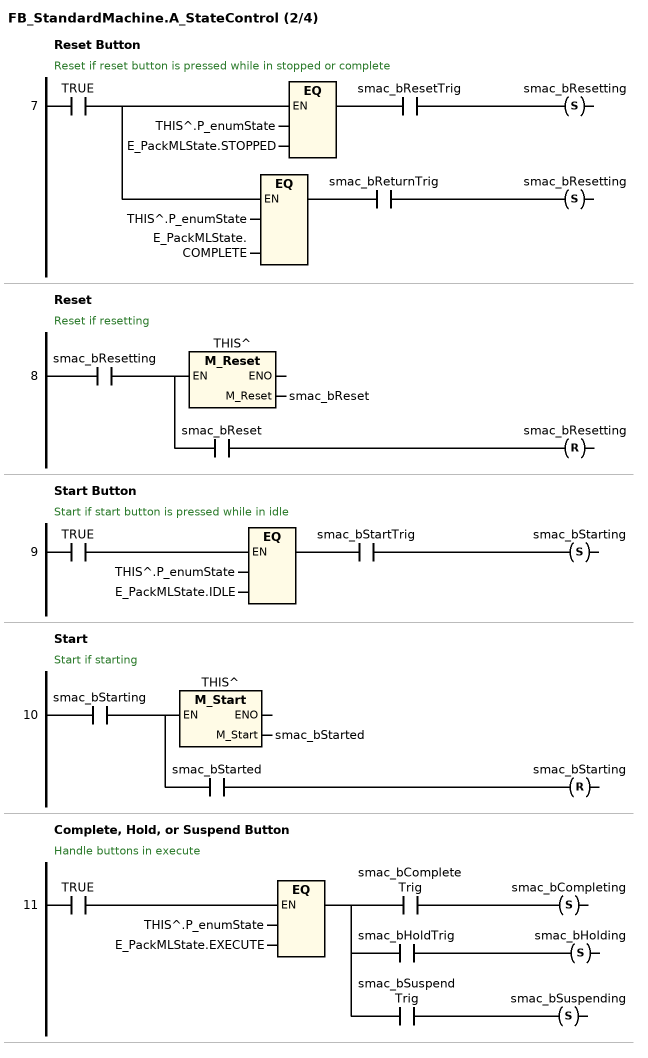
// NETWORK 7: Reset Button
// Reset if reset button is pressed while in stopped or complete
smac_bResetting S= THIS^.P_enumState = E_PackMLState.STOPPED AND smac_bResetTrig;
smac_bResetting S= THIS^.P_enumState = E_PackMLState.COMPLETE AND smac_bReturnTrig;

// NETWORK 8: Reset
// Reset if resetting
_w7 := smac_bResetting;
IF _w7 THEN THIS^.M_Reset(M_Reset => smac_bReset); END_IF
smac_bResetting R= _w7 AND smac_bReset;

// NETWORK 9: Start Button
// Start if start button is pressed while in idle
smac_bStarting S= THIS^.P_enumState = E_PackMLState.IDLE AND smac_bStartTrig;

// NETWORK 10: Start
// Start if starting
_w8 := smac_bStarting;
IF _w8 THEN THIS^.M_Start(M_Start => smac_bStarted); END_IF
smac_bStarting R= _w8 AND smac_bStarted;

// NETWORK 11: Complete, Hold, or Suspend Button
// Handle buttons in execute
_w9 := THIS^.P_enumState = E_PackMLState.EXECUTE;
smac_bCompleting S= _w9 AND smac_bCompleteTrig;
smac_bHolding S= _w9 AND smac_bHoldTrig;
smac_bSuspending S= _w9 AND smac_bSuspendTrig;

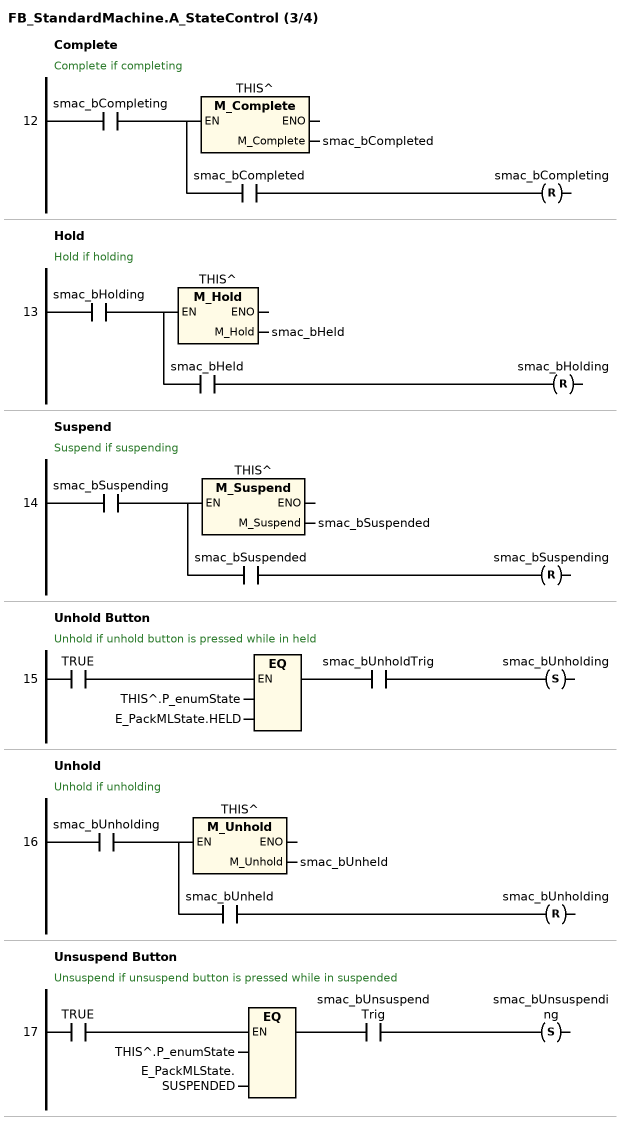
// NETWORK 12: Complete
// Complete if completing
_w10 := smac_bCompleting;
IF _w10 THEN THIS^.M_Complete(M_Complete => smac_bCompleted); END_IF
smac_bCompleting R= _w10 AND smac_bCompleted;

// NETWORK 13: Hold
// Hold if holding
_w11 := smac_bHolding;
IF _w11 THEN THIS^.M_Hold(M_Hold => smac_bHeld); END_IF
smac_bHolding R= _w11 AND smac_bHeld;

// NETWORK 14: Suspend
// Suspend if suspending
_w12 := smac_bSuspending;
IF _w12 THEN THIS^.M_Suspend(M_Suspend => smac_bSuspended); END_IF
smac_bSuspending R= _w12 AND smac_bSuspended;

// NETWORK 15: Unhold Button
// Unhold if unhold button is pressed while in held
smac_bUnholding S= THIS^.P_enumState = E_PackMLState.HELD AND smac_bUnholdTrig;

// NETWORK 16: Unhold
// Unhold if unholding
_w13 := smac_bUnholding;
IF _w13 THEN THIS^.M_Unhold(M_Unhold => smac_bUnheld); END_IF
smac_bUnholding R= _w13 AND smac_bUnheld;

// NETWORK 17: Unsuspend Button
// Unsuspend if unsuspend button is pressed while in suspended
smac_bUnsuspending S= THIS^.P_enumState = E_PackMLState.SUSPENDED AND smac_bUnsuspendTrig;

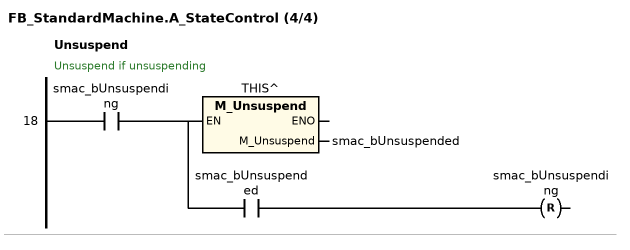
// NETWORK 18: Unsuspend
// Unsuspend if unsuspending
_w14 := smac_bUnsuspending;
IF _w14 THEN THIS^.M_Unsuspend(M_Unsuspend => smac_bUnsuspended); END_IF
smac_bUnsuspending R= _w14 AND smac_bUnsuspended;
END_ACTION

ACTION A_TrackSync:
FOR stdmac_intIndex := 1 TO UINT_TO_INT(GVL_Constants.uintMAX_MACHINE_STATION_COUNT) DO
	// Exit if pointer is not assigned
	IF mac_arrStations[stdmac_intIndex] = 0 THEN
		out_arrStationDesynched[stdmac_intIndex] := FALSE;
		CONTINUE;
	END_IF
	
	// Sync status depends on machine state
	out_arrStationDesynched[stdmac_intIndex] := TRUE;
	stdmac_enumStationState := mac_arrStations[stdmac_intIndex]^.P_enumState;
	stdmac_enumMachineState := THIS^.P_enumState;
	CASE stdmac_enumMachineState OF
		// Aborted, stopped, idle, held, suspended, or completed
		E_PackMLState.ABORTED, E_PackMLState.STOPPED, E_PackMLState.IDLE, 
				E_PackMLState.COMPLETE, E_PackMLState.HELD, E_PackMLState.SUSPENDED:
			IF stdmac_enumStationState = THIS^.P_EnumState THEN
				out_arrStationDesynched[stdmac_intIndex] := FALSE;
			END_IF
			
		// M_Abort
		E_PackMLState.ABORTING:
			CASE stdmac_enumStationState OF
				E_PackMLState.ABORTING, E_PackMLState.ABORTED:
					out_arrStationDesynched[stdmac_intIndex] := FALSE;
			END_CASE
			
		// M_Clear
		E_PackMLState.CLEARING:
			CASE stdmac_enumStationState OF
				E_PackMLState.CLEARING, E_PackMLState.STOPPED:
					out_arrStationDesynched[stdmac_intIndex] := FALSE;
			END_CASE
			
		// M_Stop
		E_PackMLState.STOPPING:
			CASE stdmac_enumStationState OF
				E_PackMLState.STOPPING, E_PackMLState.STOPPED:
					out_arrStationDesynched[stdmac_intIndex] := FALSE;
			END_CASE
			
		// M_Reset
		E_PackMLState.RESETTING:
			CASE stdmac_enumStationState OF
				E_PackMLState.RESETTING, E_PackMLState.IDLE:
					out_arrStationDesynched[stdmac_intIndex] := FALSE;
			END_CASE
			
		// M_Start
		E_PackMLState.STARTING:
			CASE stdmac_enumStationState OF
				E_PackMLState.STARTING, E_PackMLState.EXECUTE, E_PackMLState.HOLDING,
						E_PackMLState.HELD, E_PackMLState.UNHOLDING, E_PackMLState.SUSPENDING,
						E_PackMLState.SUSPENDED, E_PackMLState.UNSUSPENDING:
					out_arrStationDesynched[stdmac_intIndex] := FALSE;
			END_CASE
			
		// Execute
		E_PackMLState.EXECUTE:
			CASE stdmac_enumStationState OF
				E_PackMLState.EXECUTE, E_PackMLState.HOLDING, E_PackMLState.HELD,
						E_PackMLState.UNHOLDING, E_PackMLState.SUSPENDING,
						E_PackMLState.SUSPENDED, E_PackMLState.UNSUSPENDING:
					out_arrStationDesynched[stdmac_intIndex] := FALSE;
			END_CASE
			
		// M_Complete
		E_PackMLState.COMPLETING:
			CASE stdmac_enumStationState OF
				E_PackMLState.COMPLETING, E_PackMLState.COMPLETE:
					out_arrStationDesynched[stdmac_intIndex] := FALSE;
			END_CASE
			
		// M_Hold
		E_PackMLState.HOLDING:
			CASE stdmac_enumStationState OF
				E_PackMLState.HOLDING, E_PackMLState.HELD:
					out_arrStationDesynched[stdmac_intIndex] := FALSE;
			END_CASE
			
		// M_Unhold
		E_PackMLState.UNHOLDING:
			CASE stdmac_enumStationState OF
				E_PackMLState.EXECUTE, E_PackMLState.HOLDING, E_PackMLState.HELD,
						E_PackMLState.UNHOLDING, E_PackMLState.SUSPENDING,
						E_PackMLState.SUSPENDED, E_PackMLState.UNSUSPENDING:
					out_arrStationDesynched[stdmac_intIndex] := FALSE;
			END_CASE
			
		// M_Suspend
		E_PackMLState.SUSPENDING:
			CASE stdmac_enumStationState OF
				E_PackMLState.SUSPENDING, E_PackMLState.SUSPENDED:
					out_arrStationDesynched[stdmac_intIndex] := FALSE;
			END_CASE
			
		// M_Unsuspend
		E_PackMLState.UNSUSPENDING:
			CASE stdmac_enumStationState OF
				E_PackMLState.EXECUTE, E_PackMLState.HOLDING, E_PackMLState.HELD,
						E_PackMLState.UNHOLDING, E_PackMLState.SUSPENDING,
						E_PackMLState.SUSPENDED, E_PackMLState.UNSUSPENDING:
					out_arrStationDesynched[stdmac_intIndex] := FALSE;
			END_CASE
	END_CASE
END_FOR
END_ACTION

END_FUNCTION_BLOCK

// Interfaces/Stations/I_UserControls
INTERFACE I_UserControls

(* Clears the user prompt outputs. *)
METHOD M_ClearUserPrompt : BOOL
VAR_INPUT
END_VAR
END_METHOD

(* Sets user prompt based on given code, and awaits user input. *)
METHOD M_HandleException : BOOL
VAR_INPUT
	(* Prompt code for the exception message. *)
	_in_udintPromptCode: UDINT;
	(* Error code to set in case user aborts. *)
	_in_udintErrorCode: UDINT;
END_VAR
VAR_OUTPUT
END_VAR
END_METHOD

(* Sets out_strUserPromptCode and out_strUserPromptMessage based on
	the given user prompt code. *)
METHOD M_SetUserPrompt : BOOL
VAR_INPUT
	(* Prompt code to use for this user prompt. *)
	_in_udintCode: UDINT;
END_VAR
END_METHOD

END_INTERFACE

// Concrete/Stations/Device Test Station/FB_DeviceTestStation
FUNCTION_BLOCK FB_DeviceTestStation EXTENDS FB_SimpleStation
VAR_INPUT
	ref_fbDevice: REFERENCE TO FB_Device; // The device to be tested

	in_strProgram: T_MaxString; // Program to load when testing program loading
END_VAR
VAR_OUTPUT
	out_bAbortTested: BOOL; // Gets set to TRUE once M_Abort on ref_fbDevice has been tested once
	
	out_bConnectTested: BOOL;  // Gets set to TRUE once M_Connect on ref_fbDevice has been tested once
	out_bDisconnectTested: BOOL;  // Gets set to TRUE once M_Disconnect on ref_fbDevice has been tested once
	
	out_bEnableTested: BOOL; // Gets set to TRUE once M_Enable on ref_fbDevice has been tested once
	out_bDisableTested: BOOL; // Gets set to TRUE once M_Disable on ref_fbDevice has been tested once
	
	out_bPowerOnTested: BOOL; // Gets set to TRUE once M_PowerOn on ref_fbDevice has been tested once
	out_bPowerOffTested: BOOL; // Gets set to TRUE once M_PowerOff on ref_fbDevice has been tested once
	
	out_bLoadProgramTested: BOOL; // Gets set to TRUE once M_LoadProgram on ref_fbDevice has been tested once
	out_bStartProgramTested: BOOL; // Gets set to TRUE once M_StartProgram on ref_fbDevice has been tested once
	out_bStopProgramTested: BOOL; // Gets set to TRUE once M_StopProgram on ref_fbDevice has been tested once
	out_bPauseProgramTested: BOOL; // Gets set to TRUE once M_PauseProgram on ref_fbDevice has been tested once
	out_bUnpauseProgramTested: BOOL; // Gets set to TRUE once M_StartProgram on ref_fbDevice has been tested once after M_PauseProgram was used
	out_bStopPausedProgramTested: BOOL; // Gets set to TRUE once M_StopProgram on ref_fbDevice has been tested once after M_PauseProgram was used
	
	out_bResetTested: BOOL; // Gets set to TRUE once M_Reset on ref_fbDevice has been tested once
END_VAR
VAR
	bDeviceReset: BOOL;
	
	bDeviceConnected: BOOL;
	bDeviceDisconnected: BOOL;
	
	bDevicePoweredOn: BOOL;
	bDevicePoweredOff: BOOL;
	
	bDeviceEnabled: BOOL;
	bDeviceDisabled: BOOL;
	
	bDeviceProgramLoaded: BOOL;
	bDeviceProgramStarted: BOOL;
	bDeviceProgramStopped: BOOL;
	bDeviceProgramPaused: BOOL;

	// Device test trackers
	fbDeviceAborted: R_TRIG;
	fbDeviceReset: F_TRIG;
	fbDeviceConnected: R_TRIG;
	fbDeviceDisconnected: F_TRIG;
	fbDeviceEnabled: R_TRIG;
	fbDeviceDisabled: F_TRIG;
	fbDevicePoweredOn: R_TRIG;
	fbDevicePoweredOff: F_TRIG;
	fbDeviceProgramLoaded: R_TRIG;
	enumLastState: E_ProgramState;
END_VAR

THIS^.M_SetDevice(1, ref_fbDevice);

A_RunSimpleStation();

A_DeviceTestTracking();

ACTION A_DeviceTestTracking:
// Check device error state
fbDeviceAborted(CLK:=ref_fbDevice.P_bError);
fbDeviceReset(CLK:=ref_fbDevice.P_bError);

// Check device connection state
fbDeviceConnected(CLK:=ref_fbDevice.P_bConnected);
fbDeviceDisconnected(CLK:=ref_fbDevice.P_bConnected);

// Check device enable state
fbDeviceEnabled(CLK:=ref_fbDevice.P_bEnabled);
fbDeviceDisabled(CLK:=ref_fbDevice.P_bEnabled);

// Check device power state
fbDevicePoweredOn(CLK:=ref_fbDevice.P_bPoweredOn);
fbDevicePoweredOff(CLK:=ref_fbDevice.P_bPoweredOn);

// Check device program load state
fbDeviceProgramLoaded(CLK:=(
	ref_fbDevice.P_strCurrentProgram = in_strProgram
	AND LEN(in_strProgram) > 0));
	
// Set outputs based on triggers
IF fbDeviceAborted.Q		THEN out_bAbortTested 		:= TRUE; END_IF
IF fbDeviceReset.Q			THEN out_bResetTested 		:= TRUE; END_IF
IF fbDeviceConnected.Q		THEN out_bConnectTested 	:= TRUE; END_IF
IF fbDeviceDisconnected.Q	THEN out_bDisconnectTested	:= TRUE; END_IF
IF fbDeviceEnabled.Q		THEN out_bEnableTested 		:= TRUE; END_IF
IF fbDeviceDisabled.Q		THEN out_bDisableTested 	:= TRUE; END_IF
IF fbDevicePoweredOn.Q		THEN out_bPowerOnTested 	:= TRUE; END_IF
IF fbDevicePoweredOff.Q		THEN out_bPowerOffTested 	:= TRUE; END_IF
IF fbDeviceProgramLoaded.Q	THEN out_bLoadProgramTested	:= TRUE; END_IF

// Set program control state outputs
IF enumLastState = E_ProgramState.Stopped THEN
	IF ref_fbDevice.P_enumProgramState = E_ProgramState.Running THEN
		out_bStartProgramTested := TRUE;
	END_IF
ELSIF enumLastState = E_ProgramState.Running THEN
	IF ref_fbDevice.P_enumProgramState = E_ProgramState.Stopped THEN
		out_bStopProgramTested := TRUE;
	ELSIF ref_fbDevice.P_enumProgramState = E_ProgramState.Paused THEN
		out_bPauseProgramTested := TRUE;
	END_IF
ELSIF enumLastState = E_ProgramState.Paused THEN
	IF ref_fbDevice.P_enumProgramState = E_ProgramState.Running THEN
		out_bUnpauseProgramTested := TRUE;
	ELSIF ref_fbDevice.P_enumProgramState = E_ProgramState.Stopped THEN
		out_bStopPausedProgramTested := TRUE;
	END_IF
END_IF
enumLastState := ref_fbDevice.P_enumProgramState;
END_ACTION

END_FUNCTION_BLOCK

// Concrete/Stations/Simple Station/FB_SimpleStation
(*
	Simple station that extends adds buttons to FB_Station
*)
{attribute 'hide_all_locals'}
FUNCTION_BLOCK FB_SimpleStation EXTENDS FB_Station
VAR_INPUT
	(* Immediately abort all stations from whatever state they are in and
		go to the Aborted state. *)
	in_bAbortBtn : BOOL;
	(* Immediately stop all stations from whatever state they are in and
		go to the Stopped state. *)
	in_bStopBtn : BOOL;
	(* Clear all stations from the Aborted state and go to the Stopped state. *)
	in_bClearBtn : BOOL;
	(* Reset all stations from the Stopped state and go to the Idle state. *)
	in_bResetBtn : BOOL;
	(* Start all stations from the Idle state and go to the Execute state. *)
	in_bStartBtn : BOOL;
	(* Hold all stations from the Execute state and go to the Held state. *)
	in_bHoldBtn : BOOL;
	(* Unhold all stations from the Held state and go to the Execute state. *)
	in_bUnholdBtn : BOOL;
	(* Suspend all stations from the Execute state and go to the Held Suspended. *)
	in_bSuspendBtn : BOOL;
	(* Unsuspend all stations from the Suspended state and go to the Execute state. *)
	in_bUnsuspendBtn : BOOL;
	(* Complete all stations from the Execute state and go to the Completed state. *)
	in_bCompleteBtn : BOOL;
	(* Return all stations from the Completed state and go to the Idle state. *)
	in_bReturnBtn : BOOL;
END_VAR
VAR_OUTPUT
END_VAR
VAR
	// Abort
	ssta_fbAbortTrig: R_TRIG;
	ssta_bAbortTrig: BOOL;
	ssta_bAborting: BOOL;
	ssta_bAborted: BOOL;

	// Stop
	ssta_fbStopTrig: R_TRIG;
	ssta_bStopTrig: BOOL;
	ssta_bStopping: BOOL;
	ssta_bStopped: BOOL;
	
	// Aborted
	ssta_fbClearTrig: R_TRIG;
	ssta_bClearTrig: BOOL;
	
	// Stopped
	ssta_fbResetTrig: R_TRIG;
	ssta_bResetTrig: BOOL;
	
	// Idle
	ssta_fbStartTrig: R_TRIG;
	ssta_bStartTrig: BOOL;
	
	// Execute
	ssta_fbCompleteTrig: R_TRIG;
	ssta_bCompleteTrig: BOOL;
	ssta_fbHoldTrig: R_TRIG;
	ssta_bHoldTrig: BOOL;
	ssta_fbSuspendTrig: R_TRIG;
	ssta_bSuspendTrig: BOOL;
	
	// Complete
	ssta_fbReturnTrig: R_TRIG;
	ssta_bReturnTrig: BOOL;
	
	// Held
	ssta_fbUnholdTrig: R_TRIG;
	ssta_bUnholdTrig: BOOL;
	
	// Suspended
	ssta_fbUnsuspendTrig: R_TRIG;
	ssta_bUnsuspendTrig: BOOL;
END_VAR

THIS^.A_RunSimpleStation();

ACTION A_Buttons:
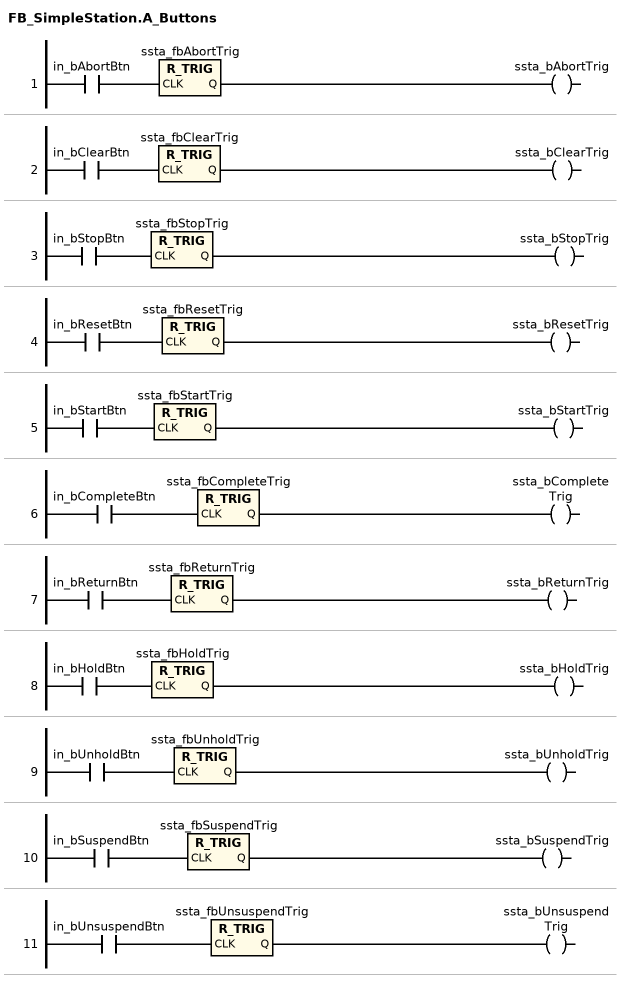
// NETWORK 1
ssta_fbAbortTrig(CLK := in_bAbortBtn); // R_TRIG
ssta_bAbortTrig := ssta_fbAbortTrig.Q;

// NETWORK 2
ssta_fbClearTrig(CLK := in_bClearBtn); // R_TRIG
ssta_bClearTrig := ssta_fbClearTrig.Q;

// NETWORK 3
ssta_fbStopTrig(CLK := in_bStopBtn); // R_TRIG
ssta_bStopTrig := ssta_fbStopTrig.Q;

// NETWORK 4
ssta_fbResetTrig(CLK := in_bResetBtn); // R_TRIG
ssta_bResetTrig := ssta_fbResetTrig.Q;

// NETWORK 5
ssta_fbStartTrig(CLK := in_bStartBtn); // R_TRIG
ssta_bStartTrig := ssta_fbStartTrig.Q;

// NETWORK 6
ssta_fbCompleteTrig(CLK := in_bCompleteBtn); // R_TRIG
ssta_bCompleteTrig := ssta_fbCompleteTrig.Q;

// NETWORK 7
ssta_fbReturnTrig(CLK := in_bReturnBtn); // R_TRIG
ssta_bReturnTrig := ssta_fbReturnTrig.Q;

// NETWORK 8
ssta_fbHoldTrig(CLK := in_bHoldBtn); // R_TRIG
ssta_bHoldTrig := ssta_fbHoldTrig.Q;

// NETWORK 9
ssta_fbUnholdTrig(CLK := in_bUnholdBtn); // R_TRIG
ssta_bUnholdTrig := ssta_fbUnholdTrig.Q;

// NETWORK 10
ssta_fbSuspendTrig(CLK := in_bSuspendBtn); // R_TRIG
ssta_bSuspendTrig := ssta_fbSuspendTrig.Q;

// NETWORK 11
ssta_fbUnsuspendTrig(CLK := in_bUnsuspendBtn); // R_TRIG
ssta_bUnsuspendTrig := ssta_fbUnsuspendTrig.Q;
END_ACTION

ACTION A_RunSimpleStation:
THIS^.A_StopAndAbort();
THIS^.A_Buttons();
THIS^.A_StateMachine();
END_ACTION

ACTION A_StopAndAbort:
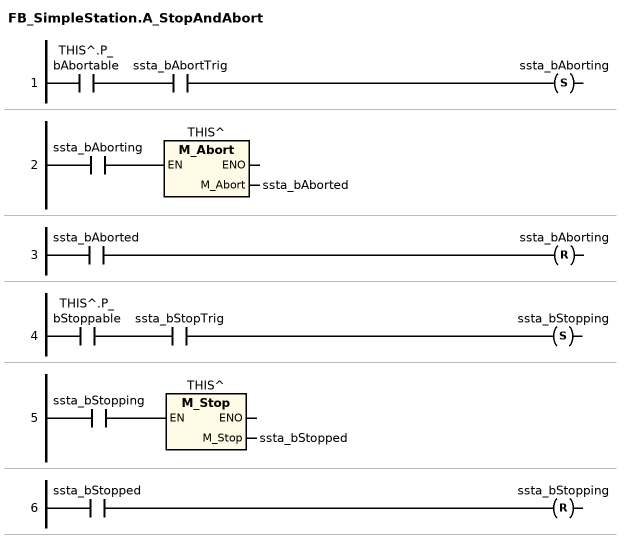
// NETWORK 1
ssta_bAborting S= THIS^.P_bAbortable AND ssta_bAbortTrig;

// NETWORK 2
IF ssta_bAborting THEN THIS^.M_Abort(M_Abort => ssta_bAborted); END_IF

// NETWORK 3
ssta_bAborting R= ssta_bAborted;

// NETWORK 4
ssta_bStopping S= THIS^.P_bStoppable AND ssta_bStopTrig;

// NETWORK 5
IF ssta_bStopping THEN THIS^.M_Stop(M_Stop => ssta_bStopped); END_IF

// NETWORK 6
ssta_bStopping R= ssta_bStopped;
END_ACTION

(* This state is entered after the aborting state completes, and should
not modify anything in the module while awaiting an explicit 'Clear' command. *)
METHOD M011_Aborted : BOOL
VAR_OUTPUT
	(* This should be set to true once an explicit 'Clear' command is received.
	Once set to true, the state machine will move to the 'Clearing' state. *)
	bClear	: BOOL;
END_VAR
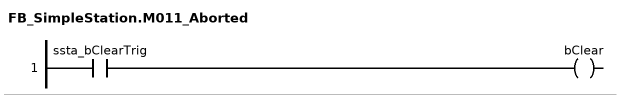
// NETWORK 1
bClear := ssta_bClearTrig;
END_METHOD

(* The machine should be stationary and awaiting an explicit 'Reset' command
while in this state. Once the 'Reset' command is received, the state machine
will move to the 'Resetting' state. *)
METHOD M111_Stopped : BOOL
VAR_OUTPUT
	(* This should be set to true if an explicit reset command is received.
	Once set to true, the state machine will move to the 'Resetting' state. *)
	bReset	: BOOL;
	(* This should be set to true if a potentially hazardous error or a safety
	fault has occurred in any tasks. Once set to true, the state machine will
	move to the 'Aborting' state. *)
	bAbort	: BOOL;
END_VAR
VAR
	_bDeviceError: BOOL;
	_strDeviceErrorId: T_MaxString;
	_udintDeviceErrorCode: UDINT;
	_strDeviceErrorMsg: T_MaxString;
	_strErrorMsg: STRING(255);
END_VAR
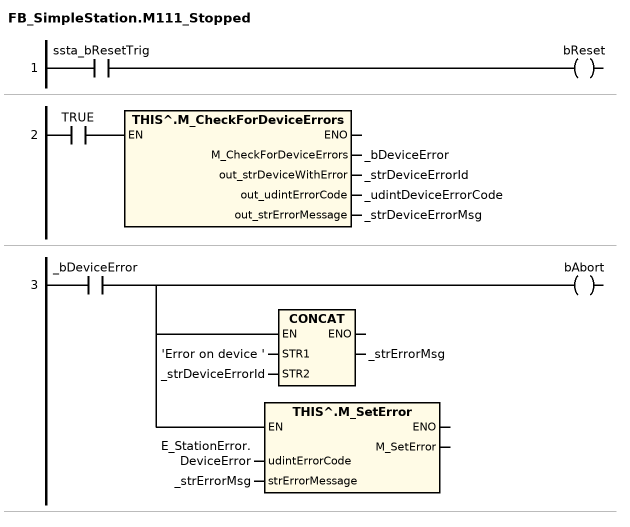
// NETWORK 1
bReset := ssta_bResetTrig;

// NETWORK 2
_bDeviceError := THIS^.M_CheckForDeviceErrors(out_strDeviceWithError => _strDeviceErrorId, out_udintErrorCode => _udintDeviceErrorCode, out_strErrorMessage => _strDeviceErrorMsg);

// NETWORK 3
bAbort := _bDeviceError;
IF _bDeviceError THEN _strErrorMsg := CONCAT(STR1 := 'Error on device ', STR2 := _strDeviceErrorId); END_IF
IF _bDeviceError THEN
    THIS^.M_SetError(udintErrorCode := E_StationError.DeviceError, strErrorMessage := _strErrorMsg);
END_IF
END_METHOD

(* This state should maintain the status of the module and its components that
was set by the resetting step while awaiting an explicit 'Start' command. *)
METHOD M211_Idle : BOOL
VAR_OUTPUT
	(* This should be set to true if an explicit 'Start' command is received.
	Once set to true, the state machine will move to the 'Starting' state. *)
	bStart	: BOOL;
	(* This should be set to true if an external source requests that the module
	exit its current state and come to a controlled stop. Once set to true, the
	state machine will move to the 'Stopping' state. *)
	bStop	: BOOL;
	(* This should be set to true if a potentially hazardous error or a safety
	fault has occurred in any tasks. Once set to true, the state machine will
	move to the 'Aborting' state. *)
	bAbort	: BOOL;
END_VAR
VAR
	_bDeviceError: BOOL;
	_strDeviceErrorId: T_MaxString;
	_udintDeviceErrorCode: UDINT;
	_strDeviceErrorMsg: T_MaxString;
	_strErrorMsg: STRING(255);
END_VAR
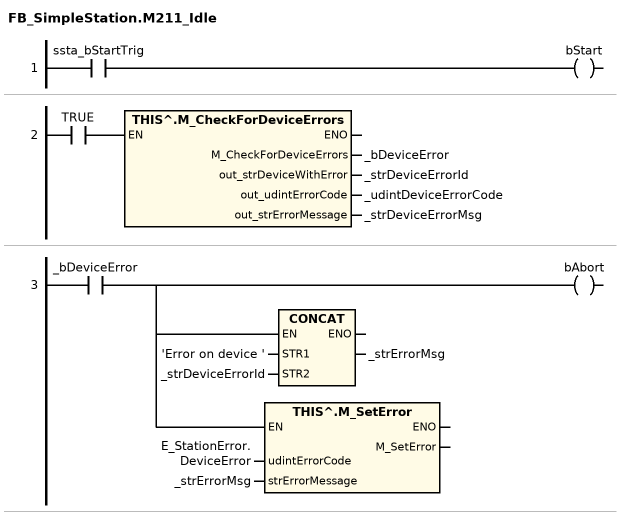
// NETWORK 1
bStart := ssta_bStartTrig;

// NETWORK 2
_bDeviceError := THIS^.M_CheckForDeviceErrors(out_strDeviceWithError => _strDeviceErrorId, out_udintErrorCode => _udintDeviceErrorCode, out_strErrorMessage => _strDeviceErrorMsg);

// NETWORK 3
bAbort := _bDeviceError;
IF _bDeviceError THEN _strErrorMsg := CONCAT(STR1 := 'Error on device ', STR2 := _strDeviceErrorId); END_IF
IF _bDeviceError THEN
    THIS^.M_SetError(udintErrorCode := E_StationError.DeviceError, strErrorMessage := _strErrorMsg);
END_IF
END_METHOD

(* The module should remain in this state while it is actively performing
automated tasks. Once all work is finished the state machine should move to the
'Completing' state. *)
METHOD M311_Execute : BOOL
VAR_OUTPUT
	(* This should be set to true once all tasks are complete and automated
	execution should be ended. Once set to true, the state machine will move to
	the 'Completing' state. *)
	bFinished	: BOOL;
	(* This should be set to true as a result of an explicit 'Hold' command
	or if internal conditions require the module to stop operation without
	completely exiting the execution sequence. Once set to true, the state
	machine will move to the 'Holding' state. *)
	bHold	: BOOL;
	(* This should be set to true if external conditions require the module to
	suspend operation until the external conditions are cleared. Once set to
	true, the state machine will move to the 'Suspending' state. *)
	bSuspend	: BOOL;
	(* This should be set to true if an external source requests that the module
	exit its current state and come to a controlled stop. Once set to true, the
	state machine will move to the 'Stopping' state. *)
	bStop	: BOOL;
	(* This should be set to true if a potentially hazardous error or a safety
	fault has occurred in any tasks. Once set to true, the state machine will
	move to the 'Aborting' state. *)
	bAbort	: BOOL;
END_VAR
VAR
	_bDeviceError: BOOL;
	_strDeviceErrorId: T_MaxString;
	_udintDeviceErrorCode: UDINT;
	_strDeviceErrorMsg: T_MaxString;
	_strErrorMsg: STRING(255);
END_VAR
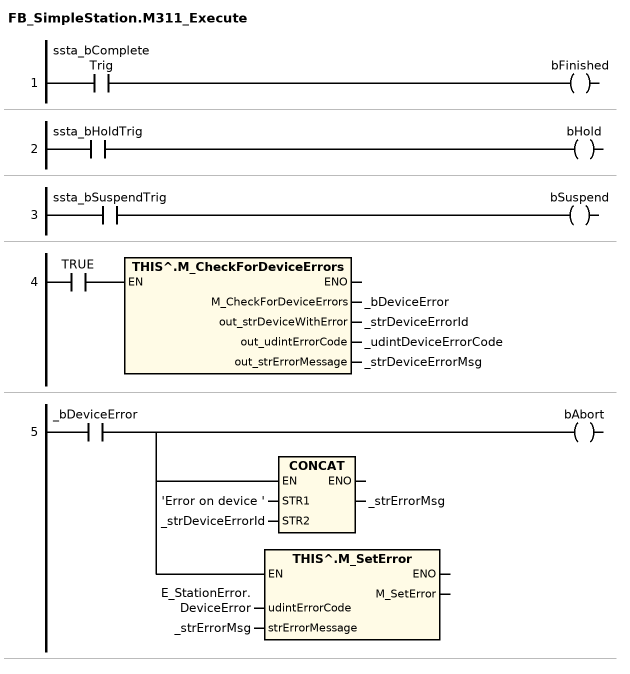
// NETWORK 1
bFinished := ssta_bCompleteTrig;

// NETWORK 2
bHold := ssta_bHoldTrig;

// NETWORK 3
bSuspend := ssta_bSuspendTrig;

// NETWORK 4
_bDeviceError := THIS^.M_CheckForDeviceErrors(out_strDeviceWithError => _strDeviceErrorId, out_udintErrorCode => _udintDeviceErrorCode, out_strErrorMessage => _strDeviceErrorMsg);

// NETWORK 5
bAbort := _bDeviceError;
IF _bDeviceError THEN _strErrorMsg := CONCAT(STR1 := 'Error on device ', STR2 := _strDeviceErrorId); END_IF
IF _bDeviceError THEN
    THIS^.M_SetError(udintErrorCode := E_StationError.DeviceError, strErrorMessage := _strErrorMsg);
END_IF
END_METHOD

(* The module should remain stationary within this state while maintaing any
execution statistics and awaiting an explicit 'Return' command. *)
METHOD M331_Complete : BOOL
VAR_OUTPUT
	(* This should be set to true if an explicit 'Return' command is received.
	Once set to true, the state machine will move to the 'Resetting' state. *)
	bReturn	: BOOL;
	(* This should be set to true if an external source requests that the module
	exit its current state and come to a controlled stop. Once set to true, the
	state machine will move to the 'Stopping' state. *)
	bStop	: BOOL;
	(* This should be set to true if a potentially hazardous error or a safety
	fault has occurred in any tasks. Once set to true, the state machine will
	move to the 'Aborting' state. *)
	bAbort	: BOOL;
END_VAR
VAR
	_bDeviceError: BOOL;
	_strDeviceErrorId: T_MaxString;
	_udintDeviceErrorCode: UDINT;
	_strDeviceErrorMsg: T_MaxString;
	_strErrorMsg: STRING(255);
END_VAR
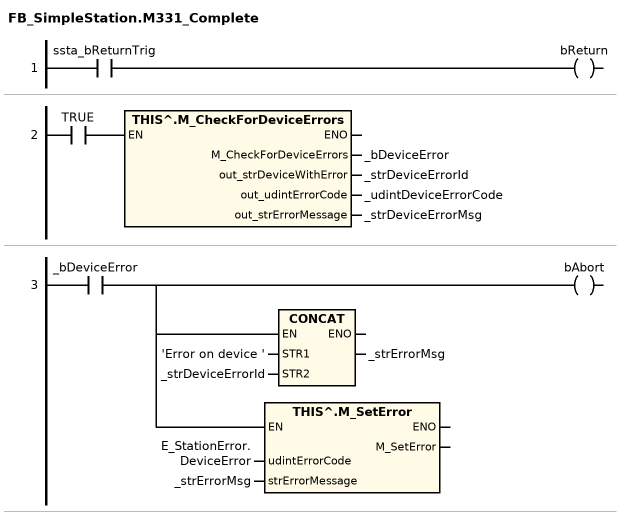
// NETWORK 1
bReturn := ssta_bReturnTrig;

// NETWORK 2
_bDeviceError := THIS^.M_CheckForDeviceErrors(out_strDeviceWithError => _strDeviceErrorId, out_udintErrorCode => _udintDeviceErrorCode, out_strErrorMessage => _strDeviceErrorMsg);

// NETWORK 3
bAbort := _bDeviceError;
IF _bDeviceError THEN _strErrorMsg := CONCAT(STR1 := 'Error on device ', STR2 := _strDeviceErrorId); END_IF
IF _bDeviceError THEN
    THIS^.M_SetError(udintErrorCode := E_StationError.DeviceError, strErrorMessage := _strErrorMsg);
END_IF
END_METHOD

(* In this state the most recent execution status should be maintained while
awaiting an explicit 'Unhold' command once internal conditions are satisfactory. *)
METHOD M411_Held : BOOL
VAR_OUTPUT
	(* This should be set to true if an explicit 'Unhold' command is received.
	Once set to true, the state machine will move to the 'Unholding' state. *)
	bUnhold	: BOOL;
	(* This should be set to true if an external source requests that the module
	exit its current state and come to a controlled stop. Once set to true, the
	state machine will move to the 'Stopping' state. *)
	bStop	: BOOL;
	(* This should be set to true if a potentially hazardous error or a safety
	fault has occurred in any tasks. Once set to true, the state machine will
	move to the 'Aborting' state. *)
	bAbort	: BOOL;
END_VAR
VAR
	_bDeviceError: BOOL;
	_strDeviceErrorId: T_MaxString;
	_udintDeviceErrorCode: UDINT;
	_strDeviceErrorMsg: T_MaxString;
	_strErrorMsg: STRING(255);
END_VAR
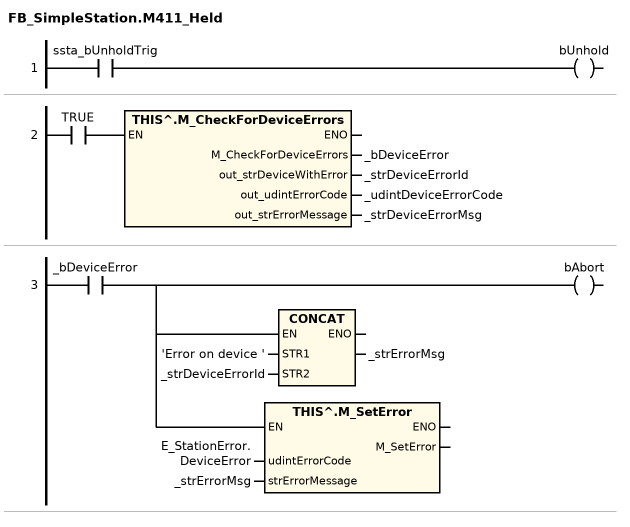
// NETWORK 1
bUnhold := ssta_bUnholdTrig;

// NETWORK 2
_bDeviceError := THIS^.M_CheckForDeviceErrors(out_strDeviceWithError => _strDeviceErrorId, out_udintErrorCode => _udintDeviceErrorCode, out_strErrorMessage => _strDeviceErrorMsg);

// NETWORK 3
bAbort := _bDeviceError;
IF _bDeviceError THEN _strErrorMsg := CONCAT(STR1 := 'Error on device ', STR2 := _strDeviceErrorId); END_IF
IF _bDeviceError THEN
    THIS^.M_SetError(udintErrorCode := E_StationError.DeviceError, strErrorMessage := _strErrorMsg);
END_IF
END_METHOD

(* In this state the most recent execution status should be maintained while
awaiting an explicit 'Unsuspend' command once external conditions are satisfactory. *)
METHOD M511_Suspended : BOOL
VAR_OUTPUT
	(* This should be set to true if an explicit 'Unsuspend' command is received.
	Once set to true, the state machine will move to the 'Unsuspending' state. *)
	bUnsuspend	: BOOL;
	(* This should be set to true if an external source requests that the module
	exit its current state and come to a controlled stop. Once set to true, the
	state machine will move to the 'Stopping' state. *)
	bStop	: BOOL;
	(* This should be set to true if a potentially hazardous error or a safety
	fault has occurred in any tasks. Once set to true, the state machine will
	move to the 'Aborting' state. *)
	bAbort	: BOOL;
END_VAR
VAR
	_bDeviceError: BOOL;
	_strDeviceErrorId: T_MaxString;
	_udintDeviceErrorCode: UDINT;
	_strDeviceErrorMsg: T_MaxString;
	_strErrorMsg: STRING(255);
END_VAR
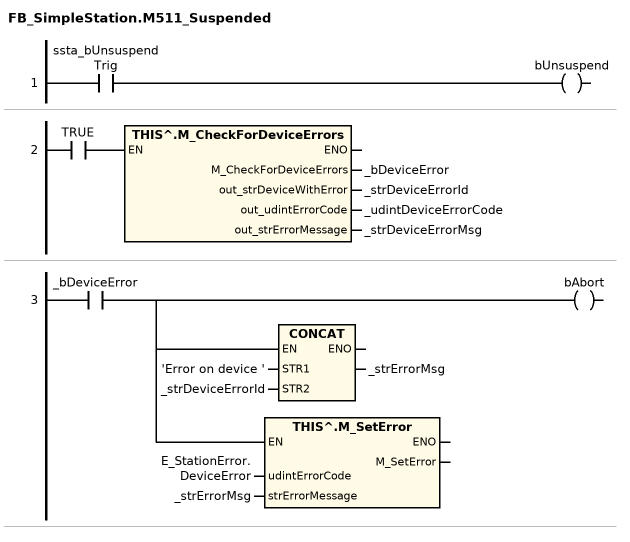
// NETWORK 1
bUnsuspend := ssta_bUnsuspendTrig;

// NETWORK 2
_bDeviceError := THIS^.M_CheckForDeviceErrors(out_strDeviceWithError => _strDeviceErrorId, out_udintErrorCode => _udintDeviceErrorCode, out_strErrorMessage => _strDeviceErrorMsg);

// NETWORK 3
bAbort := _bDeviceError;
IF _bDeviceError THEN _strErrorMsg := CONCAT(STR1 := 'Error on device ', STR2 := _strDeviceErrorId); END_IF
IF _bDeviceError THEN
    THIS^.M_SetError(udintErrorCode := E_StationError.DeviceError, strErrorMessage := _strErrorMsg);
END_IF
END_METHOD

END_FUNCTION_BLOCK

// Concrete/Stations/Remote Machine Station/FB_RemoteMachineStation
(* Function block for running a remote machine as a standard station.
	Make sure to call A_RunRemoteMachine(), which calls A_StateMachine() *)
FUNCTION_BLOCK FB_RemoteMachineStation EXTENDS FB_StandardStation 
	IMPLEMENTS I_SimpleTransitionStatesOnly, I_RemoteCycleControls
VAR CONSTANT
	rms_timeCHECK_TIME: TIME := T#1S;
	rms_timeCHECK_WAIT_TIME: TIME := T#100MS;
	rms_timeSYNC_TIME: TIME := T#1S;
END_VAR
VAR_INPUT
	(* Current remote machine state. *)
	in_enumRemoteMachineState: E_PackMLState;
	(* Remote machine error. *)
	in_bRemoteError: BOOL;
	(* Remote machine error code. *)
	in_udintRemoteErrorCode: UDINT;
	(* Ready to run signal from the remote machine. *)
	in_bRemoteReadyToRun: BOOL;
	(* Check value set by the remote machine. *)
	in_bRemoteCheckResponse: BOOL;
END_VAR
VAR_OUTPUT
	(* Run cycle command to be sent to the remote machine. *)
	out_bRemoteRunCycleCommand: BOOL;
	(* Struct of remote machine state change commands. *)
	out_stRemoteMachineCommands: ST_PackMLStateCommands;
	(* The remote machine should set in_bRemoteCheckResponse to this value to
		verify connection. *)
	out_bRemoteCheck: BOOL;
	(* TRUE if the remote machine is connected based on the remote check sequence. *)
	out_bRemoteConnected: BOOL;
END_VAR
VAR	
	rms_intRemoteCheckStep: INT;
	rms_fbCheckTimer: TON;
	rms_fbCheckWaitTimer: TON;
	rms_fbSyncTimer: TON;
	rms_enumRemoteMachineState: E_PackMLState;
	rms_enumStationState: E_PackMLState;
	rms_bRemoteMachineDesynched: BOOL;
END_VAR

A_RunRemoteMachine();

(* If the remote is ready to run, returns TRUE. *)
METHOD M_AwaitRemoteCycleEnd : BOOL
IF NOT in_bRemoteReadyToRun THEN
	out_bRemoteRunCycleCommand := FALSE;
ELSE
	M_AwaitRemoteCycleEnd := TRUE;
END_IF
END_METHOD

(* Sets run cycle command to TRUE and then waits for either the remote
	ready to run signal to get reset or for the remote to be awaiting
	end, which can happen if the remote cycle time is quicker than the
	main machine. *)
METHOD M_AwaitRemoteCycleStart : BOOL
IF in_bRemoteReadyToRun THEN
	out_bRemoteRunCycleCommand := TRUE;
ELSE
	M_AwaitRemoteCycleStart := TRUE;
END_IF
END_METHOD

METHOD M_ResetRemoteCycle : BOOL
out_bRemoteRunCycleCommand := FALSE;
END_METHOD

(* The 'Aborting' state can be entered at any time while within the 'abortable'
section of the state machine. It is typically entered in response to an 'Abort'
command or a critical fault. The logic should safely but rapidly bring the
components of the module to a stop while maintaining as much information about
the pre-abort scenario as possible. *)
METHOD M001_Aborting : BOOL
VAR_OUTPUT
	(* This should be set to true once all components of the module have safely
	come to a stop. Once set to true, the state machine will move to the
	'Aborted' state. *)
	bAborted	: BOOL;
END_VAR

VAR
	_rms_bAborted: BOOL;
END_VAR
VAR_INST // added by the converter: edge detectors and wires of the graphical bodies
    _w1 : BOOL;
END_VAR
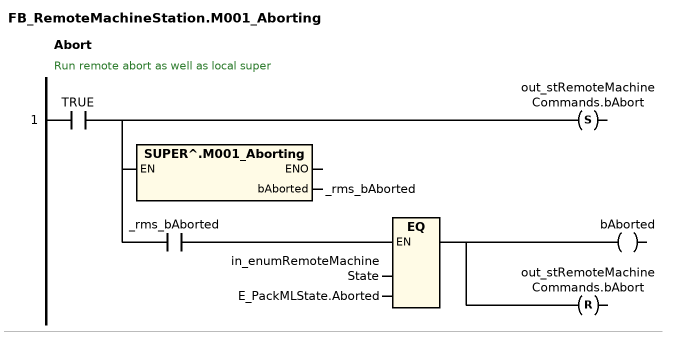
// NETWORK 1: Abort
// Run remote abort as well as local super
out_stRemoteMachineCommands.bAbort S= TRUE;
SUPER^.M001_Aborting(bAborted => _rms_bAborted);
_w1 := TRUE AND _rms_bAborted AND in_enumRemoteMachineState = E_PackMLState.Aborted;
bAborted := _w1;
out_stRemoteMachineCommands.bAbort R= _w1;
END_METHOD

(* This state should clear any faults and reset any safety features related
to the module, as well as perform actions similar to the 'Stopping' state
if they were not already performed while aborting. *)
METHOD M021_Clearing : BOOL
VAR_OUTPUT
	(* This should be set to true once the safety state of all module
	components are reset and all errors are cleared. *)
	bCleared	: BOOL;
	(* This should be set to true if a potentially hazardous error or a safety
	fault has occurred in any tasks. Once set to true, the state machine will
	move to the 'Aborting' state. *)
	bAbort	: BOOL;
END_VAR
VAR
	_rms_bCleared: BOOL;
END_VAR
VAR_INST // added by the converter: edge detectors and wires of the graphical bodies
    _w1 : BOOL;
END_VAR
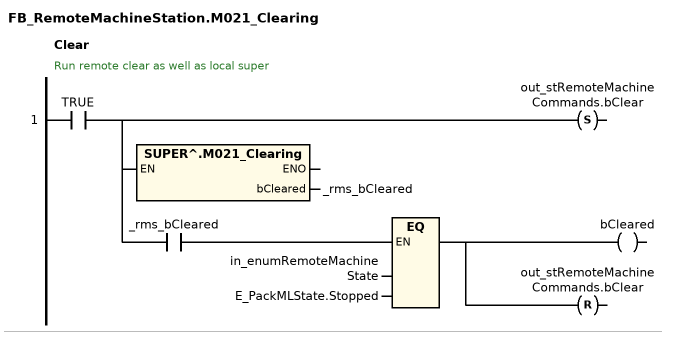
// NETWORK 1: Clear
// Run remote clear as well as local super
out_stRemoteMachineCommands.bClear S= TRUE;
SUPER^.M021_Clearing(bCleared => _rms_bCleared);
_w1 := TRUE AND _rms_bCleared AND in_enumRemoteMachineState = E_PackMLState.Stopped;
bCleared := _w1;
out_stRemoteMachineCommands.bClear R= _w1;
END_METHOD

(* This state can be entered from anywhere within the 'stoppable' group of
states. This state should safely bring the components of the module to a
controlled stop and then move to the 'Stopped' state once completed. *)
METHOD M101_Stopping : BOOL
VAR_OUTPUT
	(* This should be set to true once all relevant components have come to a
	controlled stop. Once set to true, the state machine will move to the
	'Stopped' state. *)
	bStopped	: BOOL;
	(* This should be set to true if a potentially hazardous error or a safety
	fault has occurred in any tasks. Once set to true, the state machine will
	move to the 'Aborting' state. *)
	bAbort	: BOOL;
END_VAR

VAR
	_rms_bStopped: BOOL;
END_VAR
VAR_INST // added by the converter: edge detectors and wires of the graphical bodies
    _w1 : BOOL;
END_VAR
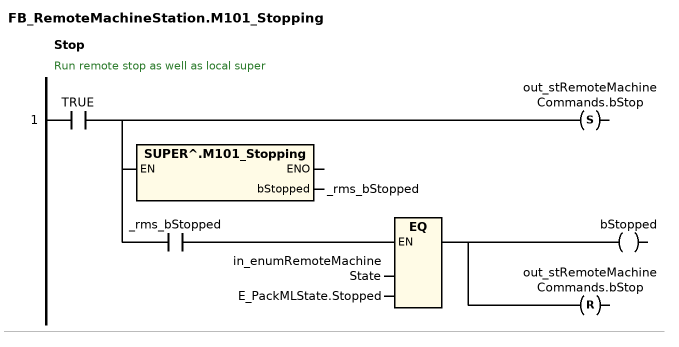
// NETWORK 1: Stop
// Run remote stop as well as local super
out_stRemoteMachineCommands.bStop S= TRUE;
SUPER^.M101_Stopping(bStopped => _rms_bStopped);
_w1 := TRUE AND _rms_bStopped AND in_enumRemoteMachineState = E_PackMLState.Stopped;
bStopped := _w1;
out_stRemoteMachineCommands.bStop R= _w1;
END_METHOD

(* This state should place the module and all of its components into a safe
energized idle state where it will wait for a start command. Once all tasks are
complete, it will move to the 'Idle' state. No external movement should occur
as a result of this state. *)
METHOD M201_Resetting : BOOL
VAR_OUTPUT
	(* Set this to true once the module is energized and ready to start.
	Once set to true, the state machine will move to the 'Idle' state. *)
	bIdle	: BOOL;
	(* This should be set to true if an external source requests that the module
	exit its current state and come to a controlled stop. Once set to true, the
	state machine will move to the 'Stopping' state. *)
	bStop	: BOOL;
	(* This should be set to true if a potentially hazardous error or a safety
	fault has occurred in any tasks. Once set to true, the state machine will
	move to the 'Aborting' state. *)
	bAbort	: BOOL;
END_VAR

VAR
	_rms_bIdle: BOOL;
END_VAR
VAR_INST // added by the converter: edge detectors and wires of the graphical bodies
    _w1 : BOOL;
END_VAR
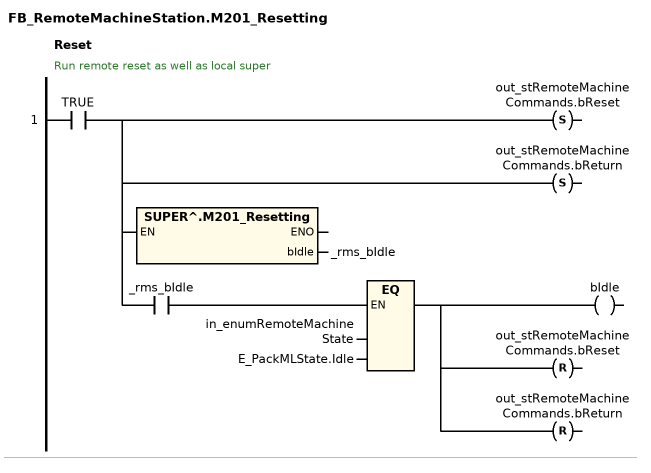
// NETWORK 1: Reset
// Run remote reset as well as local super
out_stRemoteMachineCommands.bReset S= TRUE;
out_stRemoteMachineCommands.bReturn S= TRUE;
SUPER^.M201_Resetting(bIdle => _rms_bIdle);
_w1 := TRUE AND _rms_bIdle AND in_enumRemoteMachineState = E_PackMLState.Idle;
bIdle := _w1;
out_stRemoteMachineCommands.bReset R= _w1;
out_stRemoteMachineCommands.bReturn R= _w1;
END_METHOD

(* This state should make any final preparations needed for the 'Execute' state
prior to entering the 'Execute' state. *)
METHOD M301_Starting : BOOL
VAR_OUTPUT
	(* This should be set to true once the module and its components are fully
	prepared for process execution. Once set to true, the state machine will
	move to the 'Execute' state. *)
	bStarted	: BOOL;
	(* This should be set to true if an external source requests that the module
	exit its current state and come to a controlled stop. Once set to true, the
	state machine will move to the 'Stopping' state. *)
	bStop	: BOOL;
	(* This should be set to true if a potentially hazardous error or a safety
	fault has occurred in any tasks. Once set to true, the state machine will
	move to the 'Aborting' state. *)
	bAbort	: BOOL;
END_VAR

VAR
	_rms_bStarted: BOOL;
END_VAR
VAR_INST // added by the converter: edge detectors and wires of the graphical bodies
    _w1 : BOOL;
END_VAR
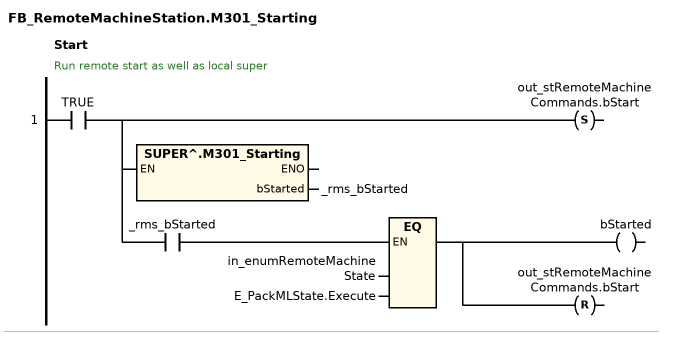
// NETWORK 1: Start
// Run remote start as well as local super
out_stRemoteMachineCommands.bStart S= TRUE;
SUPER^.M301_Starting(bStarted => _rms_bStarted);
_w1 := TRUE AND _rms_bStarted AND in_enumRemoteMachineState = E_PackMLState.Execute;
bStarted := _w1;
out_stRemoteMachineCommands.bStart R= _w1;
END_METHOD

(* This state will perform any post-execution tasks prior to moving to the
'Completed' state. *)
METHOD M321_Completing : BOOL
VAR_OUTPUT
	(* Move to the Complete state*)
	bCompleted	: BOOL;
	(* This should be set to true if an external source requests that the module
	exit its current state and come to a controlled stop. Once set to true, the
	state machine will move to the 'Stopping' state. *)
	bStop	: BOOL;
	(* This should be set to true if a potentially hazardous error or a safety
	fault has occurred in any tasks. Once set to true, the state machine will
	move to the 'Aborting' state. *)
	bAbort	: BOOL;
END_VAR

VAR
	_rms_bCompleted: BOOL;
END_VAR
VAR_INST // added by the converter: edge detectors and wires of the graphical bodies
    _w1 : BOOL;
END_VAR
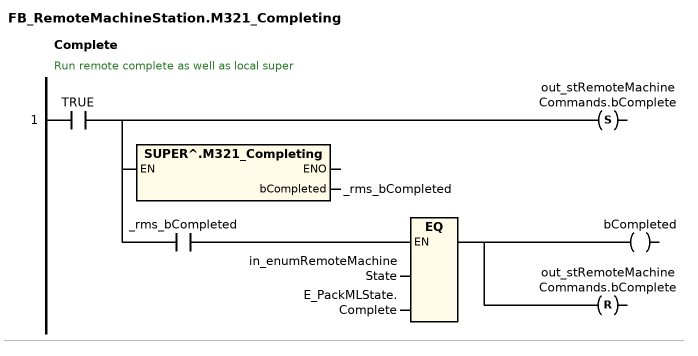
// NETWORK 1: Complete
// Run remote complete as well as local super
out_stRemoteMachineCommands.bComplete S= TRUE;
SUPER^.M321_Completing(bCompleted => _rms_bCompleted);
_w1 := TRUE AND _rms_bCompleted AND in_enumRemoteMachineState = E_PackMLState.Complete;
bCompleted := _w1;
out_stRemoteMachineCommands.bComplete R= _w1;
END_METHOD

(* This state should safely pause task executions without completely ending or
resetting them. *)
METHOD M401_Holding : BOOL
VAR_OUTPUT
	(* This should be set to true once all execution tasks are safely paused.
	Once set to true, the state machine will move to the 'Held' state. *)
	bHeld	: BOOL;
	(* This should be set to true if an external source requests that the module
	exit its current state and come to a controlled stop. Once set to true, the
	state machine will move to the 'Stopping' state. *)
	bStop	: BOOL;
	(* This should be set to true if a potentially hazardous error or a safety
	fault has occurred in any tasks. Once set to true, the state machine will
	move to the 'Aborting' state. *)
	bAbort	: BOOL;
END_VAR

VAR
	_rms_bHeld: BOOL;
END_VAR
VAR_INST // added by the converter: edge detectors and wires of the graphical bodies
    _w1 : BOOL;
END_VAR
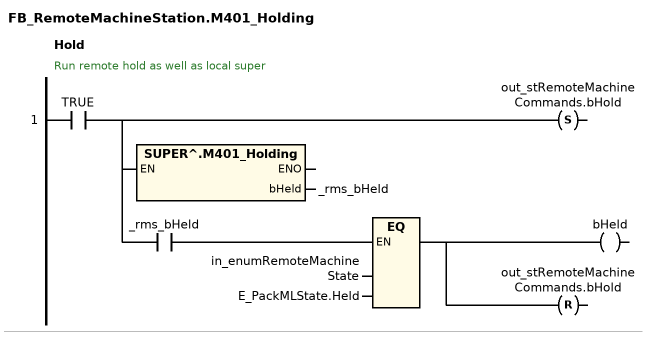
// NETWORK 1: Hold
// Run remote hold as well as local super
out_stRemoteMachineCommands.bHold S= TRUE;
SUPER^.M401_Holding(bHeld => _rms_bHeld);
_w1 := TRUE AND _rms_bHeld AND in_enumRemoteMachineState = E_PackMLState.Held;
bHeld := _w1;
out_stRemoteMachineCommands.bHold R= _w1;
END_METHOD

(* In this state, the module and its components should be returned to the
scenario it was in before it entered the 'Holding' step so that the
'Execute' state can pick up where it left off. *)
METHOD M421_Unholding : BOOL
VAR_OUTPUT
	(* This should be set to true once the module is ready to restart
	execution. Once set to true, the state machine will move to the 'Execute'
	state. *)
	bUnheld	: BOOL;
	(* This should be set to true if an external source requests that the module
	exit its current state and come to a controlled stop. Once set to true, the
	state machine will move to the 'Stopping' state. *)
	bStop	: BOOL;
	(* This should be set to true if a potentially hazardous error or a safety
	fault has occurred in any tasks. Once set to true, the state machine will
	move to the 'Aborting' state. *)
	bAbort	: BOOL;
END_VAR

VAR
	_rms_bUnheld: BOOL;
END_VAR
VAR_INST // added by the converter: edge detectors and wires of the graphical bodies
    _w1 : BOOL;
END_VAR
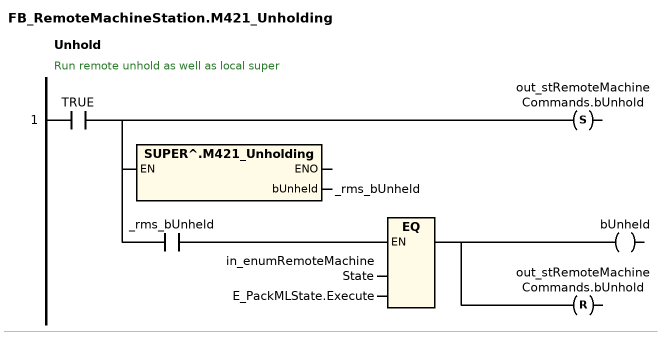
// NETWORK 1: Unhold
// Run remote unhold as well as local super
out_stRemoteMachineCommands.bUnhold S= TRUE;
SUPER^.M421_Unholding(bUnheld => _rms_bUnheld);
_w1 := TRUE AND _rms_bUnheld AND in_enumRemoteMachineState = E_PackMLState.Execute;
bUnheld := _w1;
out_stRemoteMachineCommands.bUnhold R= _w1;
END_METHOD

(* This state should safely pause task executions without completely ending or
resetting them. *)
METHOD M501_Suspending : BOOL
VAR_OUTPUT
	(* This should be set to true once all execution tasks are safely paused.
	Once set to true, the state machine will move to the 'Suspended' state. *)
	bSuspended	: BOOL;
	(* This should be set to true if an external source requests that the module
	exit its current state and come to a controlled stop. Once set to true, the
	state machine will move to the 'Stopping' state. *)
	bStop	: BOOL;
	(* This should be set to true if a potentially hazardous error or a safety
	fault has occurred in any tasks. Once set to true, the state machine will
	move to the 'Aborting' state. *)
	bAbort	: BOOL;
END_VAR

VAR
	_rms_bSuspended: BOOL;
END_VAR
VAR_INST // added by the converter: edge detectors and wires of the graphical bodies
    _w1 : BOOL;
END_VAR
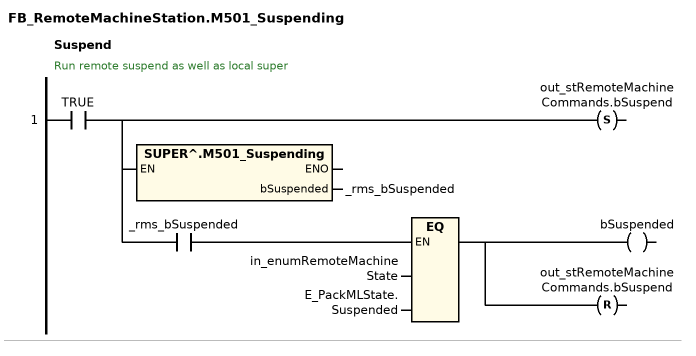
// NETWORK 1: Suspend
// Run remote suspend as well as local super
out_stRemoteMachineCommands.bSuspend S= TRUE;
SUPER^.M501_Suspending(bSuspended => _rms_bSuspended);
_w1 := TRUE AND _rms_bSuspended AND in_enumRemoteMachineState = E_PackMLState.Suspended;
bSuspended := _w1;
out_stRemoteMachineCommands.bSuspend R= _w1;
END_METHOD

(* In this state, the module and its components should be returned to the
scenario it was in before it entered the 'Suspending' step so that the
'Execute' state can pick up where it left off. *)
METHOD M521_Unsuspending : BOOL
VAR_OUTPUT
	(* This should be set to true once the module is ready to restart
	execution. Once set to true, the state machine will move to the 'Execute'
	state. *)
	bUnsuspended	: BOOL;
	(* This should be set to true if an external source requests that the module
	exit its current state and come to a controlled stop. Once set to true, the
	state machine will move to the 'Stopping' state. *)
	bStop	: BOOL;
	(* This should be set to true if a potentially hazardous error or a safety
	fault has occurred in any tasks. Once set to true, the state machine will
	move to the 'Aborting' state. *)
	bAbort	: BOOL;
END_VAR

VAR
	_rms_bUnsuspended: BOOL;
END_VAR
VAR_INST // added by the converter: edge detectors and wires of the graphical bodies
    _w1 : BOOL;
END_VAR
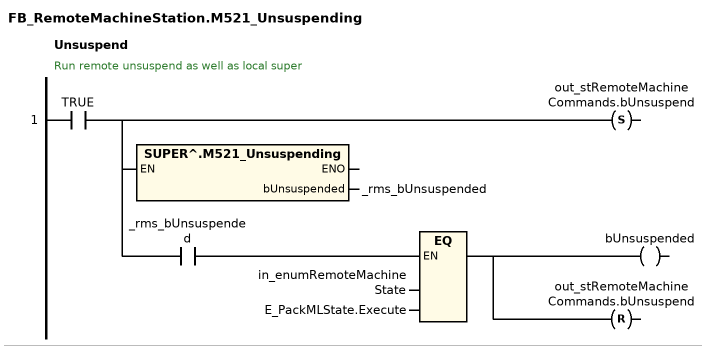
// NETWORK 1: Unsuspend
// Run remote unsuspend as well as local super
out_stRemoteMachineCommands.bUnsuspend S= TRUE;
SUPER^.M521_Unsuspending(bUnsuspended => _rms_bUnsuspended);
_w1 := TRUE AND _rms_bUnsuspended AND in_enumRemoteMachineState = E_PackMLState.Execute;
bUnsuspended := _w1;
out_stRemoteMachineCommands.bUnsuspend R= _w1;
END_METHOD

ACTION A_RemoteCheck:
CASE rms_intRemoteCheckStep OF
	0:	// Initialize
		rms_fbCheckTimer(IN:=FALSE);
		out_bRemoteCheck := TRUE;
		rms_intRemoteCheckStep := 10;
	10: // Wait for response
		IF in_bRemoteCheckResponse = out_bRemoteCheck THEN
			out_bRemoteConnected := TRUE;
			rms_fbCheckWaitTimer(IN:=FALSE);
			rms_intRemoteCheckStep := 20;
		ELSE
			rms_fbCheckTimer(IN:=TRUE, PT:=rms_timeCHECK_TIME);
			IF rms_fbCheckTimer.Q THEN
				out_bRemoteConnected := FALSE;
			END_IF
		END_IF
	20: // Change output
		rms_fbCheckWaitTimer(IN:=TRUE, PT:=rms_timeCHECK_WAIT_TIME);
		IF rms_fbCheckWaitTimer.Q THEN
			rms_fbCheckTimer(IN:=FALSE);
			out_bRemoteCheck := NOT out_bRemoteCheck;
			rms_intRemoteCheckStep := 10;
		END_IF
END_CASE
END_ACTION

ACTION A_RemoteSync:
// Sync status depends on state
rms_bRemoteMachineDesynched := TRUE;
rms_enumRemoteMachineState := in_enumRemoteMachineState;
rms_enumStationState := THIS^.P_enumState;
CASE rms_enumStationState OF
	// Aborted, stopped, idle, execute, held, suspended, or completed
	E_PackMLState.ABORTED, E_PackMLState.STOPPED, E_PackMLState.IDLE, E_PackMLState.EXECUTE,
			E_PackMLState.COMPLETE, E_PackMLState.HELD, E_PackMLState.SUSPENDED:
		IF rms_enumRemoteMachineState = THIS^.P_EnumState THEN
			rms_fbSyncTimer(IN:=FALSE);
			rms_bRemoteMachineDesynched := FALSE;
		END_IF
		
	// M_Abort
	E_PackMLState.ABORTING:
		CASE rms_enumRemoteMachineState OF
			E_PackMLState.ABORTING, E_PackMLState.ABORTED:
				rms_fbSyncTimer(IN:=FALSE);
				rms_bRemoteMachineDesynched := FALSE;
		ELSE
			IF out_stRemoteMachineCommands.bAbort THEN
				rms_fbSyncTimer(IN:=TRUE, PT:=rms_timeSYNC_TIME);
				IF NOT rms_fbSyncTimer.Q THEN
					rms_bRemoteMachineDesynched := FALSE;
				END_IF
			ELSE
				rms_bRemoteMachineDesynched := FALSE;
			END_IF
		END_CASE
		
	// M_Clear
	E_PackMLState.CLEARING:
		CASE rms_enumRemoteMachineState OF
			E_PackMLState.CLEARING, E_PackMLState.STOPPED:
				rms_fbSyncTimer(IN:=FALSE);
				rms_bRemoteMachineDesynched := FALSE;
			E_PackMLState.ABORTED:
				IF out_stRemoteMachineCommands.bClear THEN
					rms_fbSyncTimer(IN:=TRUE, PT:=rms_timeSYNC_TIME);
					IF NOT rms_fbSyncTimer.Q THEN
						rms_bRemoteMachineDesynched := FALSE;
					END_IF
				ELSE
					rms_bRemoteMachineDesynched := FALSE;
				END_IF
		END_CASE
		
	// M_Stop
	E_PackMLState.STOPPING:
		CASE rms_enumRemoteMachineState OF
			E_PackMLState.STOPPING, E_PackMLState.STOPPED:
				rms_fbSyncTimer(IN:=FALSE);
				rms_bRemoteMachineDesynched := FALSE;
			E_PackMLState.ABORTING, E_PackMLState.ABORTED, E_PackMLState.CLEARING:
				rms_bRemoteMachineDesynched := TRUE;
		ELSE
			IF out_stRemoteMachineCommands.bStop THEN
				rms_fbSyncTimer(IN:=TRUE, PT:=rms_timeSYNC_TIME);
				IF NOT rms_fbSyncTimer.Q THEN
					rms_bRemoteMachineDesynched := FALSE;
				END_IF
			ELSE
				rms_bRemoteMachineDesynched := FALSE;
			END_IF
		END_CASE
		
	// M_Reset
	E_PackMLState.RESETTING:
		CASE rms_enumRemoteMachineState OF
			E_PackMLState.RESETTING, E_PackMLState.IDLE:
				rms_fbSyncTimer(IN:=FALSE);
				rms_bRemoteMachineDesynched := FALSE;
			E_PackMLState.STOPPED:
				IF out_stRemoteMachineCommands.bReset THEN
					rms_fbSyncTimer(IN:=TRUE, PT:=rms_timeSYNC_TIME);
					IF NOT rms_fbSyncTimer.Q THEN
						rms_bRemoteMachineDesynched := FALSE;
					END_IF
				ELSE
					rms_bRemoteMachineDesynched := FALSE;
				END_IF
			E_PackMLState.COMPLETE:
				IF out_stRemoteMachineCommands.bReturn THEN
					rms_fbSyncTimer(IN:=TRUE, PT:=rms_timeSYNC_TIME);
					IF NOT rms_fbSyncTimer.Q THEN
						rms_bRemoteMachineDesynched := FALSE;
					END_IF
				ELSE
					rms_bRemoteMachineDesynched := FALSE;
				END_IF
		END_CASE
		
	// M_Start
	E_PackMLState.STARTING:
		CASE rms_enumRemoteMachineState OF
			E_PackMLState.STARTING, E_PackMLState.EXECUTE:
				rms_fbSyncTimer(IN:=FALSE);
				rms_bRemoteMachineDesynched := FALSE;
			E_PackMLState.IDLE:
				IF out_stRemoteMachineCommands.bStart THEN
					rms_fbSyncTimer(IN:=TRUE, PT:=rms_timeSYNC_TIME);
					IF NOT rms_fbSyncTimer.Q THEN
						rms_bRemoteMachineDesynched := FALSE;
					END_IF
				ELSE
					rms_bRemoteMachineDesynched := FALSE;
				END_IF
		END_CASE
		
	// M_Complete
	E_PackMLState.COMPLETING:
		CASE rms_enumRemoteMachineState OF
			E_PackMLState.COMPLETING, E_PackMLState.COMPLETE:
				rms_fbSyncTimer(IN:=FALSE);
				rms_bRemoteMachineDesynched := FALSE;
			E_PackMLState.EXECUTE:
				IF out_stRemoteMachineCommands.bComplete THEN
					rms_fbSyncTimer(IN:=TRUE, PT:=rms_timeSYNC_TIME);
					IF NOT rms_fbSyncTimer.Q THEN
						rms_bRemoteMachineDesynched := FALSE;
					END_IF
				ELSE
					rms_bRemoteMachineDesynched := FALSE;
				END_IF
		END_CASE
		
	// M_Hold
	E_PackMLState.HOLDING:
		CASE rms_enumRemoteMachineState OF
			E_PackMLState.HOLDING, E_PackMLState.HELD:
				rms_fbSyncTimer(IN:=FALSE);
				rms_bRemoteMachineDesynched := FALSE;
			E_PackMLState.EXECUTE:
				IF out_stRemoteMachineCommands.bHold THEN
					rms_fbSyncTimer(IN:=TRUE, PT:=rms_timeSYNC_TIME);
					IF NOT rms_fbSyncTimer.Q THEN
						rms_bRemoteMachineDesynched := FALSE;
					END_IF
				ELSE
					rms_bRemoteMachineDesynched := FALSE;
				END_IF
		END_CASE
		
	// M_Unhold
	E_PackMLState.UNHOLDING:
		CASE rms_enumRemoteMachineState OF
			E_PackMLState.UNHOLDING, E_PackMLState.EXECUTE:
				rms_fbSyncTimer(IN:=FALSE);
				rms_bRemoteMachineDesynched := FALSE;
			E_PackMLState.HELD:
				IF out_stRemoteMachineCommands.bUnhold THEN
					rms_fbSyncTimer(IN:=TRUE, PT:=rms_timeSYNC_TIME);
					IF NOT rms_fbSyncTimer.Q THEN
						rms_bRemoteMachineDesynched := FALSE;
					END_IF
				ELSE
					rms_bRemoteMachineDesynched := FALSE;
				END_IF
		END_CASE
		
	// M_Suspend
	E_PackMLState.SUSPENDING:
		CASE rms_enumRemoteMachineState OF
			E_PackMLState.SUSPENDING, E_PackMLState.SUSPENDED:
				rms_fbSyncTimer(IN:=FALSE);
				rms_bRemoteMachineDesynched := FALSE;
			E_PackMLState.EXECUTE:
				IF out_stRemoteMachineCommands.bSuspend THEN
					rms_fbSyncTimer(IN:=TRUE, PT:=rms_timeSYNC_TIME);
					IF NOT rms_fbSyncTimer.Q THEN
						rms_bRemoteMachineDesynched := FALSE;
					END_IF
				ELSE
					rms_bRemoteMachineDesynched := FALSE;
				END_IF
		END_CASE
		
	// M_Unsuspend
	E_PackMLState.UNSUSPENDING:
		CASE rms_enumRemoteMachineState OF
			E_PackMLState.UNSUSPENDING, E_PackMLState.EXECUTE:
				rms_fbSyncTimer(IN:=FALSE);
				rms_bRemoteMachineDesynched := FALSE;
			E_PackMLState.SUSPENDED:
				IF out_stRemoteMachineCommands.bUnsuspend THEN
					rms_fbSyncTimer(IN:=TRUE, PT:=rms_timeSYNC_TIME);
					IF NOT rms_fbSyncTimer.Q THEN
						rms_bRemoteMachineDesynched := FALSE;
					END_IF
				ELSE
					rms_bRemoteMachineDesynched := FALSE;
				END_IF
		END_CASE
END_CASE

// Move to remote machine state if desynched and connected
IF out_bRemoteConnected AND rms_bRemoteMachineDesynched THEN
	THIS^.M_MoveToState(in_enumRemoteMachineState);
END_IF
END_ACTION

ACTION A_RunRemoteMachine:
THIS^.A_StateMachine();
IF NOT in_bDisableStateMethods THEN
	THIS^.A_RemoteCheck();
	THIS^.A_RemoteSync();
END_IF
//IF in_bRemoteError THEN
//	THIS^.M_SetError(in_udintRemoteErrorCode, 'Remote machine had an error!');
//END_IF
END_ACTION

END_FUNCTION_BLOCK

// Concrete/Stations/Standard Station/FB_StandardStation
(*
===============================================================================
Standard Station
===============================================================================
:Contact: Kevin Sanita <ksanita@sensata.com>
:Last Edited: February 2023

:Description: The standard station adds a number of common station functionalities
	such as waiting for cycle start/stop, handling exceptions and user prompts,
	and collecting general statistics about cycles.

:Notes:
* The cycle controls are M_AwaitCycleStart, M_AwaitCycleEnd, and M_ResetCycle.
	- M_AwaitCycleStart will set out_bReadyToRun to TRUE and wait for
		in_bRunCycleCommand to be TRUE before setting out_bReadyToRun to FALSE
		and returning TRUE.
	- M_AwaitCycleEnd will set out_bReadyToRun to TRUE and wait for
		in_bRunCycleCommand to be FALSE before returning TRUE.
	- M_ResetCycle will set out_bReadyToRun to FALSE. This is important in
		scenarios such as when the station aborts while still awaiting cycle end.
* The user controls are M_SetUserPrompt, M_ClearUserPrompt, and M_HandleException.
	- M_SetUserPrompt takes in a user prompt code and sets the relevant
		user prompt from in_arrUserPrompts, sets out_udintUserPromptCode and
		out_strUserPromptMessage, and logs the user message.
	- M_ClearUserPrompt just clears the active user prompt
	- M_HandleException takes in a user prompt code and an error code, and then
		awaits one of in_bUserRetry or in_bUserAbort to be set to TRUE. If
		in_bUserRetry is set to TRUE, M_HandleException will return TRUE.
		IF in_bUserAbort is set to TRUE, an error will be set on the station
		with the given error code.
* The only method for cycle statistics is M_ResetCycleStatistics, which will clear
	the current statistics. Otherwise all the various statistics are stored as
	properties, and relate to the cycle controls. Any statistics with "Cycle"
	measure from M_AwaitCycleStart=TRUE to the first call of M_AwaitCycleEnd,
	and any statistics with "Wait" measure the time between cycles. Utilization
	is a measure of "Cycle" time / total time. 

:Change Log:
- **February 2023** Initial version (K. Sanita)
- **May 2023** Added cycle statistics (K. Sanita)
*)
FUNCTION_BLOCK FB_StandardStation EXTENDS FB_Station IMPLEMENTS I_CycleControls, I_CycleStatistics, I_UserControls
VAR CONSTANT
	(* This is here for backwards compatibility. Use GVL_Constants.intMAX_USER_PROMPTS instead. *)
	intMAX_USER_PROMPTS : INT := GVL_Constants.intMAX_USER_PROMPTS;
END_VAR
VAR_INPUT
	(* Station will start running process cycle once this is set to
		TRUE, and then will wait for this to be set to FALSE before
		resetting back to initial step. *)
	in_bRunCycleCommand: BOOL;
	(* Array of user prompts. *)
	in_arrUserPrompts: ARRAY[1..GVL_Constants.intMAX_USER_PROMPTS] OF ST_Prompt;
	(* User retry signal for an exception state. *)
	in_bUserRetry: BOOL;
	(* User stop machine signal for an exception state. *)
	in_bUserAbort: BOOL;
END_VAR
VAR_OUTPUT
	(* Station should set this to TRUE while the process cycle is
		not running, and FALSE while running. *)
	out_bReadyToRun: BOOL;
	(* ID of the current user prompt. *)
	out_udintUserPromptCode: UDINT;
	(* Default message of the current user prompt. *)
	out_strUserPromptMessage: T_MaxString;
END_VAR
VAR
	ssta_ulintCycleStartTime: ULINT;
	ssta_ulintCycleEndTime: ULINT;
	ssta_udintCycleCount: UDINT;
	ssta_lrealLastCycleTime: LREAL;
	ssta_lrealAvgCycleTime: LREAL;
	ssta_bCycleComplete: BOOL;
	
	ssta_ulintWaitStartTime: ULINT;
	ssta_ulintWaitEndTime: ULINT;
	ssta_udintWaitCount: UDINT;
	ssta_lrealLastWaitTime: LREAL;
	ssta_lrealAvgWaitTime: LREAL;
	ssta_bWaitComplete: BOOL;
	
	ssta_lrealLastUtilization: LREAL;
	ssta_lrealAvgUtilization: LREAL;
	
	ssta_bAwaitingStart: BOOL;
	ssta_bAwaitingEnd: BOOL;
END_VAR

(* Sets ready to run to TRUE and waits for run cycle command to be reset. *)
METHOD M_AwaitCycleEnd : BOOL
VAR_INPUT
END_VAR

VAR
	_lrealStartTime: LREAL;
	_lrealEndTime: LREAL;
	
END_VAR
VAR_INST
	_inst_lrealAvgCycleTime: LREAL;
	_inst_bCycleComplete: BOOL;
END_VAR
M_AwaitCycleEnd := FALSE;
ssta_bAwaitingStart := FALSE;
ssta_bAwaitingEnd := TRUE;

IF NOT _inst_bCycleComplete THEN
	THIS^.M_LogMessage('Cycle complete.');
	ssta_ulintWaitStartTime := F_GetSystemTime();
	ssta_ulintCycleEndTime := F_GetSystemTime();

	IF ssta_ulintCycleStartTime > 0 THEN
		_lrealStartTime := ULINT_TO_LREAL(ssta_ulintCycleStartTime / 10) / 1000000;
		_lrealEndTime := ULINT_TO_LREAL(ssta_ulintCycleEndTime / 10) / 1000000;
		ssta_lrealLastCycleTime := _lrealEndTime - _lrealStartTime;
		IF NOT ssta_bCycleComplete THEN
			_inst_lrealAvgCycleTime := ssta_lrealAvgCycleTime;
			ssta_udintCycleCount := ssta_udintCycleCount + 1;
			ssta_bCycleComplete := TRUE;
			ssta_bWaitComplete := FALSE;
		END_IF
		ssta_lrealAvgCycleTime := ((ssta_udintCycleCount - 1) * _inst_lrealAvgCycleTime + ssta_lrealLastCycleTime) / (ssta_udintCycleCount);
		IF (ssta_lrealAvgCycleTime + ssta_lrealAvgWaitTime) > 0 THEN
			ssta_lrealAvgUtilization := ssta_lrealAvgCycleTime / (ssta_lrealAvgCycleTime + ssta_lrealAvgWaitTime);
		END_IF
		IF (ssta_lrealLastCycleTime + ssta_lrealLastWaitTime) > 0 THEN
			ssta_lrealLastUtilization := ssta_lrealLastCycleTime / (ssta_lrealLastCycleTime + ssta_lrealLastWaitTime);
		END_IF
	END_IF
END_IF
_inst_bCycleComplete := TRUE;

IF NOT in_bRunCycleCommand THEN
	_inst_bCycleComplete := FALSE;
	out_bReadyToRun := TRUE;
	M_AwaitCycleEnd := TRUE;
	ssta_bAwaitingEnd := FALSE;
END_IF
END_METHOD

(* Sets ready to run to TRUE and then waits for run cycle command. *)
METHOD M_AwaitCycleStart : BOOL
VAR_INPUT
END_VAR

VAR
	_lrealStartTime: LREAL;
	_lrealEndTime: LREAL;
END_VAR
VAR_INST
	_inst_lrealAvgWaitTime: LREAL;
END_VAR
M_AwaitCycleStart := FALSE;
ssta_bAwaitingStart := TRUE;
ssta_bAwaitingEnd := FALSE;

out_bReadyToRun := TRUE;
IF in_bRunCycleCommand THEN
	out_bReadyToRun := FALSE;
	M_AwaitCycleStart := TRUE;
	ssta_bAwaitingStart := FALSE;
	ssta_ulintCycleStartTime := F_GetSystemTime();
	ssta_ulintWaitEndTime := F_GetSystemTime();
	
	IF ssta_ulintWaitStartTime > 0 THEN
		_lrealStartTime := ULINT_TO_LREAL(ssta_ulintWaitStartTime / 10) / 1000000;
		_lrealEndTime := ULINT_TO_LREAL(ssta_ulintWaitEndTime / 10) / 1000000;
		ssta_lrealLastWaitTime := _lrealEndTime - _lrealStartTime;
		IF NOT ssta_bWaitComplete THEN
			_inst_lrealAvgWaitTime := ssta_lrealAvgWaitTime;
			ssta_udintWaitCount := ssta_udintWaitCount + 1;
			ssta_bWaitComplete := TRUE;
			ssta_bCycleComplete := FALSE;
		END_IF
		ssta_lrealAvgWaitTime := ((ssta_udintWaitCount - 1) * _inst_lrealAvgWaitTime + ssta_lrealLastWaitTime) / (ssta_udintWaitCount);
	END_IF
END_IF
END_METHOD

METHOD M_ResetCycle : BOOL
VAR_INPUT
END_VAR
out_bReadyToRun := FALSE;
ssta_ulintCycleStartTime := 0;
ssta_ulintCycleEndTime := 0;
ssta_ulintWaitStartTime := 0;
ssta_ulintWaitEndTime := 0;
ssta_bCycleComplete := FALSE;
ssta_bWaitComplete := FALSE;
M_ResetCycle := TRUE;
ssta_bAwaitingStart := FALSE;
ssta_bAwaitingEnd := FALSE;
END_METHOD

PROPERTY P_bAwaitingEnd : BOOL
GET
P_bAwaitingEnd := ssta_bAwaitingEnd;
END_GET
END_PROPERTY

PROPERTY P_bAwaitingStart : BOOL
GET
P_bAwaitingStart := ssta_bAwaitingStart;
END_GET
END_PROPERTY

METHOD M_ResetCycleStatistics : BOOL
VAR_INPUT
END_VAR
ssta_ulintCycleStartTime:=0;
ssta_ulintCycleEndTime:=0;
ssta_udintCycleCount:=0;
ssta_lrealLastCycleTime:=0;
ssta_lrealAvgCycleTime:=0;

ssta_ulintWaitStartTime:=0;
ssta_ulintWaitEndTime:=0;
ssta_udintWaitCount:=0;
ssta_lrealLastWaitTime:=0;
ssta_lrealAvgWaitTime:=0;

ssta_lrealLastUtilization:=0;
ssta_lrealAvgUtilization:=0;
END_METHOD

PROPERTY P_lrealAvgCycleTime : LREAL
GET
P_lrealAvgCycleTime := ssta_lrealAvgCycleTime;
END_GET
END_PROPERTY

PROPERTY P_lrealAvgUtilization : LREAL
GET
P_lrealAvgUtilization := ssta_lrealAvgUtilization;
END_GET
END_PROPERTY

PROPERTY P_lrealAvgWaitTime : LREAL
GET
P_lrealAvgWaitTime := ssta_lrealAvgWaitTime;
END_GET
END_PROPERTY

PROPERTY P_lrealLastCycleTime : LREAL
GET
P_lrealLastCycleTime := ssta_lrealLastCycleTime;
END_GET
END_PROPERTY

PROPERTY P_lrealLastUtilization : LREAL
GET
P_lrealLastUtilization := ssta_lrealLastUtilization;
END_GET
END_PROPERTY

PROPERTY P_lrealLastWaitTime : LREAL
GET
P_lrealLastWaitTime := ssta_lrealLastWaitTime;
END_GET
END_PROPERTY

PROPERTY P_udintCycleCount : UDINT
GET
P_udintCycleCount := ssta_udintCycleCount;
END_GET
END_PROPERTY

PROPERTY P_udintWaitCount : UDINT
GET
P_udintWaitCount := ssta_udintWaitCount;
END_GET
END_PROPERTY

(* Clears the user prompt outputs. *)
METHOD M_ClearUserPrompt : BOOL
VAR_INPUT
END_VAR
out_strUserPromptMessage := '';
out_udintUserPromptCode := 0;
M_ClearUserPrompt := TRUE;
END_METHOD

(* Sets user prompt based on given code, and awaits user input. *)
METHOD M_HandleException : BOOL
VAR_INPUT
	(* Prompt code for the exception message. *)
	_in_udintPromptCode: UDINT;
	(* Error code to set in case user aborts. *)
	_in_udintErrorCode: UDINT;
END_VAR
VAR_OUTPUT
END_VAR
M_HandleException := FALSE;
THIS^.M_SetUserPrompt(_in_udintPromptCode);
IF in_bUserRetry THEN
	THIS^.M_ClearUserPrompt();
	M_HandleException := TRUE;
ELSIF in_bUserAbort THEN
	THIS^.M_SetError(_in_udintErrorCode, 'User chose to abort after an exception.');
END_IF
END_METHOD

(* Sets out_strUserPromptCode and out_strUserPromptMessage based on
	the given user prompt code. *)
METHOD M_SetUserPrompt : BOOL
VAR_INPUT
	(* Prompt code to use for this user prompt. *)
	_in_udintCode: UDINT;
END_VAR

VAR
	_strMessage: T_MaxString;
	_intIndex: INT;
END_VAR
FOR _intIndex := 1 TO GVL_Constants.intMAX_USER_PROMPTS DO
	IF in_arrUserPrompts[_intIndex].udintCode = _in_udintCode THEN
		_strMessage := in_arrUserPrompts[_intIndex].strMessage;
		EXIT;
	END_IF
END_FOR
IF out_udintUserPromptCode <> _in_udintCode THEN
	IF LEN(_strMessage) > 0 THEN
		THIS^.M_LogMessage(_strMessage);
	ELSE
		THIS^.M_LogWarning('Prompt message not found!');
	END_IF
END_IF
out_strUserPromptMessage := _strMessage;
out_udintUserPromptCode := _in_udintCode;
M_SetUserPrompt := TRUE;
END_METHOD

END_FUNCTION_BLOCK

// Interfaces/Stations/I_CycleControls
INTERFACE I_CycleControls

(* Sets ready to run to TRUE and waits for run cycle command to be reset. *)
METHOD M_AwaitCycleEnd : BOOL
VAR_INPUT
END_VAR
END_METHOD

(* Sets ready to run to TRUE and then waits for run cycle command. *)
METHOD M_AwaitCycleStart : BOOL
VAR_INPUT
END_VAR
END_METHOD

METHOD M_ResetCycle : BOOL
VAR_INPUT
END_VAR
END_METHOD

PROPERTY P_bAwaitingEnd : BOOL
GET
END_GET
END_PROPERTY

PROPERTY P_bAwaitingStart : BOOL
GET
END_GET
END_PROPERTY

END_INTERFACE

// Interfaces/Stations/I_CycleStatistics
INTERFACE I_CycleStatistics

METHOD M_ResetCycleStatistics : BOOL
VAR_INPUT
END_VAR
END_METHOD

PROPERTY P_lrealAvgCycleTime : LREAL
GET
END_GET
END_PROPERTY

PROPERTY P_lrealAvgUtilization : LREAL
GET
END_GET
END_PROPERTY

PROPERTY P_lrealAvgWaitTime : LREAL
GET
END_GET
END_PROPERTY

PROPERTY P_lrealLastCycleTime : LREAL
GET
END_GET
END_PROPERTY

PROPERTY P_lrealLastUtilization : LREAL
GET
END_GET
END_PROPERTY

PROPERTY P_lrealLastWaitTime : LREAL
GET
END_GET
END_PROPERTY

PROPERTY P_udintCycleCount : UDINT
GET
END_GET
END_PROPERTY

PROPERTY P_udintWaitCount : UDINT
GET
END_GET
END_PROPERTY

END_INTERFACE

// Interfaces/Stations/I_RemoteCycleControls
(* Used if a remote machine or station has multiple cycles per local station cycle. *)
INTERFACE I_RemoteCycleControls

(* Sets ready to run to TRUE and waits for run cycle command to be reset. *)
METHOD M_AwaitRemoteCycleEnd : BOOL
VAR_INPUT
END_VAR
END_METHOD

(* Sets ready to run to TRUE and then waits for run cycle command. *)
METHOD M_AwaitRemoteCycleStart : BOOL
VAR_INPUT
END_VAR
END_METHOD

METHOD M_ResetRemoteCycle : BOOL
VAR_INPUT
END_VAR
END_METHOD

END_INTERFACE

// Interfaces/Devices/I_Triggerable
INTERFACE I_Triggerable

(* Triggers an action  on the device used such as marking,printing, welding, cleaning, etc. *)
METHOD M_Trigger : BOOL
VAR_INPUT
END_VAR
END_METHOD

END_INTERFACE

// Interfaces/Modules/I_Cyclic
INTERFACE I_Cyclic

METHOD M_RunModule : BOOL
VAR_INPUT
END_VAR
END_METHOD

END_INTERFACE

// Interfaces/State Machine/Stateful/I_ExecuteStateOnly
(* This interface only implements the methods for the Execute state. *)
INTERFACE I_ExecuteStateOnly EXTENDS I_SimpleExecuteStateOnly

(* Runs for a single cycle when entering the execute state. *)
METHOD M310_Execute_Entry : BOOL
VAR_INPUT
END_VAR
END_METHOD

(* Runs for a single cycle when exiting the execute state. *)
METHOD M312_Execute_Exit : BOOL
VAR_INPUT
END_VAR
END_METHOD

END_INTERFACE

// Interfaces/Stations/I_StationDeviceControl
INTERFACE I_StationDeviceControl

(* Aborts all devices set in the station. *)
METHOD M_AbortDevices : BOOL
VAR_INPUT
END_VAR
END_METHOD

(* Clears all devices set in the station. *)
METHOD M_ClearDevices : BOOL
VAR_INPUT
END_VAR
END_METHOD

(* Completes all devices set in the station. *)
METHOD M_CompleteDevices : BOOL
VAR_INPUT
END_VAR
END_METHOD

(* Holds all devices set in the station. *)
METHOD M_HoldDevices : BOOL
VAR_INPUT
END_VAR
END_METHOD

(* Resets all devices set in the station. *)
METHOD M_ResetDevices : BOOL
VAR_INPUT
END_VAR
END_METHOD

(* Starts all devices set in the station. *)
METHOD M_StartDevices : BOOL
VAR_INPUT
END_VAR
END_METHOD

(* Stops all devices set in the station. *)
METHOD M_StopDevices : BOOL
VAR_INPUT
END_VAR
END_METHOD

(* Suspends all devices set in the station. *)
METHOD M_SuspendDevices : BOOL
VAR_INPUT
END_VAR
END_METHOD

(* Unholds all devices set in the station. *)
METHOD M_UnholdDevices : BOOL
VAR_INPUT
END_VAR
END_METHOD

(* Unsuspends all devices set in the station. *)
METHOD M_UnsuspendDevices : BOOL
VAR_INPUT
END_VAR
END_METHOD

END_INTERFACE

// Project Information/F_GetCompany
// This function has been automatically generated from the project information.
{attribute 'signature_flag' := '1073741824'}
{attribute 'TcGenerated'}
{attribute 'no-analysis'}
FUNCTION F_GetCompany : WSTRING
VAR_INPUT
	
END_VAR

F_GetCompany := "Sensata Technologies";

END_FUNCTION

// Project Information/F_GetTitle
// This function has been automatically generated from the project information.
{attribute 'signature_flag' := '1073741824'}
{attribute 'TcGenerated'}
{attribute 'no-analysis'}
FUNCTION F_GetTitle : WSTRING
VAR_INPUT
	
END_VAR

F_GetTitle := "Sensata_Common";

END_FUNCTION

// Project Information/F_GetVersion
// This function has been automatically generated from the project information.
{attribute 'signature_flag' := '1073741824'}
{attribute 'TcGenerated'}
{attribute 'no-analysis'}
FUNCTION F_GetVersion : ST_LibVersion
VAR_INPUT
	
END_VAR

F_GetVersion.iMajor := 3;
F_GetVersion.iMinor := 0;
F_GetVersion.iBuild := 4;
F_GetVersion.iRevision := 0;
F_GetVersion.sVersion := '3.0.4';
F_GetVersion.nFlags := 0;

END_FUNCTION
